FUNCTION_BLOCK FB_Example
VAR
    iValue : INT;
END_VAR
BEGIN
iResult := iValue + iRes;
END_FUNCTION_BLOCK
